{region '#Template'}
	{attribute 'Version' := '0.0.1.0'}
	{attribute 'Tags' := '"LCID": "1031", "Text": "General, Settings, Project, Basics"'}
	{attribute 'Tags' := '"LCID": "1033", "Text": "General, Settings, Project, Basics"'}
	{attribute 'Description' := '"LCID": "1031", "Text": "Basis Einstellungen der Steuerung, system services"'}
	{attribute 'Description' := '"LCID": "1033", "Text": "Basic settings of the control"'}
{endregion}
FUNCTION_BLOCK FB_BA_IFP EXTENDS FB_BA_View
VAR_INPUT
END_VAR
VAR_INPUT CONSTANT
	Project							: FB_BA_ProjectEx := (nInstanceID				:= 12345);
	Trend							: FB_BA_TrendLogging;	
END_VAR
VAR_OUTPUT
END_VAR
VAR
//	LblAggregates.AutomationStationEquipment
//	LblControl.BACnetDevice
	LblProject			:FB_BA_Label2x :=(iAggregate:=LblAggregates.AutomationStationEquipment,	 iFunction:=LblControl.BACnetDevice);	
END_VAR

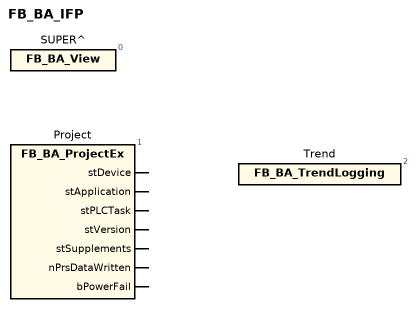
SUPER^(); // FB_BA_View
Project(); // FB_BA_ProjectEx
Trend(); // FB_BA_TrendLogging

METHOD FB_init : BOOL
VAR_INPUT
	bInitRetains : BOOL; // if TRUE, the retain variables are initialized (warm start / cold start)
	bInCopyCode : BOOL;  // if TRUE, the instance afterwards gets moved into the copy code (online change)
END_VAR
Project.iParent					:= THIS^;
Project.iLabel					:= LblProject;
//	Project.sObjectName				:= LblProject;		
//	Project.sDescription			:= 'Projektinformationen';
//	Project.nInstanceID				:= 12345;

Trend.iParent					:= THIS^;
Trend.iLabel					:= LblControl.TrendLogging;
Trend.sObjectName				:= '{Idx=01}';
Trend.eDPADMode					:= E_BA_DPADMode.eInclude;
END_METHOD

END_FUNCTION_BLOCK

(* stored: Version 1.1.0.1, ProductVersion 3.1.4024.6
   POU FB_BA_IFP: Id {d4b2b7cd-0261-4932-97f0-e657fec2866c}, SpecialFunc None
   Method FB_init: Id {a6ea51b1-fc25-4891-bcad-ddbebe33c60e} *)
